GLOBALCONSTANTS NVS_Keys (* Global constants *)
  (* Standard: 61499-1 *)
  (* Version 1.0, 2024-02-25, franz *)
  VAR_GLOBAL CONSTANT
    KEY_I1_STORE : STRING := 'K_I1';
  END_VAR
END_GLOBALCONSTANTS
